{attribute 'linkalways'}
{attribute 'hide_all_locals'}
FUNCTION_BLOCK ValueLreal EXTENDS ValueLrealRead IMPLEMENTS Value
VAR
END_VAR

METHOD Set : BOOL
VAR_INPUT
	source : ANY;
END_VAR
Set := ConvertAnyType(source, thisAnyType);
END_METHOD

METHOD SetFromString : BOOL
VAR_INPUT
	value : T_MaxString;
END_VAR
thisValue := STRING_TO_LREAL(value);

SetFromString := TRUE;
END_METHOD

METHOD SetFromType : BOOL
VAR_INPUT
	source : __SYSTEM.AnyType;
END_VAR
SetFromType := ConvertAnyType(source, thisAnyType);
END_METHOD

END_FUNCTION_BLOCK

(* stored: Version 1.1.0.1, ProductVersion 3.1.4024.15
   POU ValueLreal: Id {b7b078d1-e9d0-4fd9-8a17-f8630bb0b52f}, SpecialFunc None
   Method Set: Id {13bc8491-1df9-43a8-a775-82e554a66250}
   Method SetFromString: Id {b7de7043-b32b-4e78-83d1-fdb44e57e319}
   Method SetFromType: Id {d8e29480-2cb5-4487-a342-5b14a745bc95} *)
